// TIA Portal V20 export
// export: Created 2026-09-14T11:29:51.0854813Z, ExportSetting None, DisplayName Totally Integrated Automation Portal, DisplayVersion V20, DisplayName TIA Portal Openness, DisplayVersion V20, DisplayName TIA Portal Version Control Interface, DisplayVersion V20, DisplayName STEP 7 Professional, DisplayVersion V20, DisplayName STEP 7 Safety, DisplayVersion V20, DisplayName WinCC Basic/Comfort/Advanced, DisplayVersion V20, DisplayName WinCC Unified, DisplayVersion V20
VAR_GLOBAL   // PLC tag table "TrafficLightTags"
   northLightGreen AT %Q0.0 : Bool;
   northLightYellow AT %Q0.1 : Bool;
   northLightRed AT %Q0.2 : Bool;
   southLightGreen AT %Q0.3 : Bool;
   southLightYellow AT %Q0.4 : Bool;
   southLightRed AT %Q0.5 : Bool;
   eastLightGreen AT %Q1.0 : Bool;
   eastLightYellow AT %Q1.1 : Bool;
   eastLightRed AT %Q1.2 : Bool;
   westLightGreen AT %Q1.3 : Bool;
   westLightYellow AT %Q1.4 : Bool;
   westLightRed AT %Q1.5 : Bool;
   systemFAULT AT %M2.0 : Bool;
   start_MEM_TAG AT %M2.2 : Bool;
   reset_MEM_TAG AT %M2.1 : Bool;
   start_Button_IN AT %I0.0 : Bool;
   reset_Button_IN AT %I0.1 : Bool;
END_VAR
